FUNCTION_BLOCK CAT_Robotino (* Composite Function Block Type *)
  (* Standard: 61499-2 *)
  (* Version 0.0, 26/10/2022, Pranay Jhunjhunwala, Schneider Electric, template *)
  PACKAGE Main;
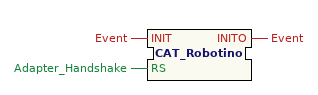
  EVENT_INPUT
    INIT; (* Initialization Request *)
  END_EVENT
  EVENT_OUTPUT
    INITO; (* Initialization Confirm *)
  END_EVENT
  SOCKETS
    RS : Adapter_Handshake;
  END_SOCKETS
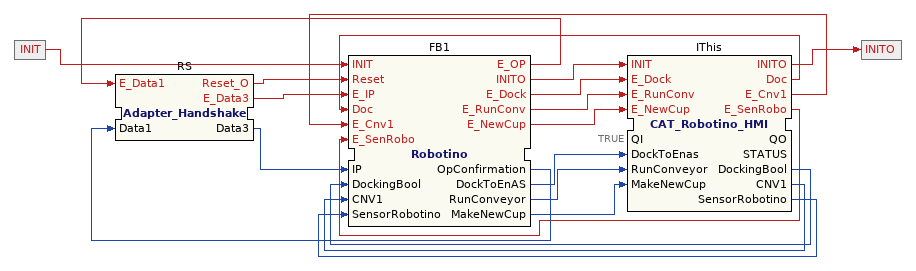
  FBS
    FB1 : Robotino;
    IThis : CAT_Robotino_HMI(QI := TRUE);
  END_FBS
  EVENT_CONNECTIONS
    INIT TO FB1.INIT;
    RS.Reset_O TO FB1.Reset;
    RS.E_Data3 TO FB1.E_IP;
    FB1.E_OP TO RS.E_Data1;
    FB1.INITO TO IThis.INIT;
    FB1.E_Dock TO IThis.E_Dock;
    FB1.E_RunConv TO IThis.E_RunConv;
    FB1.E_NewCup TO IThis.E_NewCup;
    IThis.INITO TO INITO;
    IThis.Doc TO FB1.Doc;
    IThis.E_Cnv1 TO FB1.E_Cnv1;
    IThis.E_SenRobo TO FB1.E_SenRobo;
  END_CONNECTIONS
  DATA_CONNECTIONS
    RS.Data3 TO FB1.IP;
    FB1.OpConfirmation TO RS.Data1;
    FB1.DockToEnAS TO IThis.DockToEnas;
    FB1.RunConveyor TO IThis.RunConveyor;
    FB1.MakeNewCup TO IThis.MakeNewCup;
    IThis.DockingBool TO FB1.DockingBool;
    IThis.CNV1 TO FB1.CNV1;
    IThis.SensorRobotino TO FB1.SensorRobotino;
  END_CONNECTIONS
END_FUNCTION_BLOCK
